// Tests for MONETRoof.FB_Roof's state machine (code review finding L5).
//
// Covers: the E_RoofState.unknown default before the first call, opening/closing (driven purely by
// Open()/Close()/SoftStop() and the ramp, no hardware inputs needed), stopped, and Reset() recovering
// from a cleared error.
//
// Deliberately not covered: the opened/closed states. Both need roof_limit_open/roof_limit_closed,
// which come from motors[i].opened/.closed -- AT%I*, hardware-linked, and this project configures no
// I/O. Validate those on the PLC instead (same as the plan's open step 5).
//
// Two things every test here has to do (without them FB_Roof never leaves the error / stopped state):
//  - SetDrivesOk(): FB_RoofMotor.motor_error is AT%I* and means "drive OK" (error := NOT motor_error). This project
//    maps no I/O, so it stays FALSE and both motors report error, which puts FB_Roof into the error state.
//  - one Call() before Open()/Close(): FB_Roof's parameters (max_speed, ...) are VAR_INPUTs that are only assigned
//    by a call, so Open() before the first call sets target_speed := TO_INT(0).
FUNCTION_BLOCK FB_Roof_State_Tests EXTENDS TcUnit.FB_TestSuite
VAR
END_VAR

Initial_State_Is_Unknown();
Open_Drives_State_To_Opening();
SoftStop_From_Moving_Drives_State_To_Stopped();
Close_Drives_State_To_Closing();
Reset_Clears_Error_State();

METHOD PRIVATE Call
VAR_IN_OUT
	roof		: MONETRoof.FB_Roof;
END_VAR
VAR_INPUT
	comm		: BROTLib.I_Comm;
END_VAR
roof(
	roof_number			:= 1,
	min_speed			:= 10000,
	max_speed			:= 30000,
	acceleration		:= 150,
	min_position		:= 0,
	max_position		:= 200,
	max_position_diff	:= 2,
	comm				:= comm);
END_METHOD

METHOD PRIVATE SetDrivesOk
VAR_IN_OUT
	roof		: MONETRoof.FB_Roof;
END_VAR
// motor_error is AT%I* with no I/O mapped here: TRUE = drive OK (see the header comment)
roof.motors[1].motor_error := TRUE;
roof.motors[2].motor_error := TRUE;
END_METHOD

METHOD PRIVATE Initial_State_Is_Unknown
VAR
	fbRoof	: MONETRoof.FB_Roof;
END_VAR
// Before FB_Roof is ever called, its VAR_OUTPUT members already hold their declared defaults.
TEST('Initial_State_Is_Unknown');
AssertTrue(Condition := fbRoof.state = E_RoofState.unknown, Message := 'declared default before the first call (was closed / enum value 0, L5)');
TEST_FINISHED();
END_METHOD

METHOD PRIVATE Open_Drives_State_To_Opening
VAR
	fbRoof	: MONETRoof.FB_Roof;
	fbComm	: FB_NullComm;
END_VAR
TEST('Open_Drives_State_To_Opening');
SetDrivesOk(roof := fbRoof);
Call(roof := fbRoof, comm := fbComm);	// assigns the parameters; Open() before this would see max_speed = 0
fbRoof.Open();
Call(roof := fbRoof, comm := fbComm);
AssertTrue(Condition := fbRoof.state = E_RoofState.opening, Message := 'speed > 0, both motors moving and direction_open: state becomes opening');
TEST_FINISHED();
END_METHOD

METHOD PRIVATE SoftStop_From_Moving_Drives_State_To_Stopped
VAR
	fbRoof	: MONETRoof.FB_Roof;
	fbComm	: FB_NullComm;
END_VAR
TEST('SoftStop_From_Moving_Drives_State_To_Stopped');
SetDrivesOk(roof := fbRoof);
Call(roof := fbRoof, comm := fbComm);	// assigns the parameters
fbRoof.Open();
Call(roof := fbRoof, comm := fbComm);
AssertTrue(Condition := fbRoof.state = E_RoofState.opening, Message := 'sanity: moving before the stop');
fbRoof.SoftStop();
// speed was 150, accel is 150: one ramp step reaches exactly 0
Call(roof := fbRoof, comm := fbComm);
AssertTrue(Condition := fbRoof.state = E_RoofState.stopped, Message := 'ramped down to 0, no longer moving, no switches engaged: stopped');
TEST_FINISHED();
END_METHOD

METHOD PRIVATE Close_Drives_State_To_Closing
VAR
	fbRoof	: MONETRoof.FB_Roof;
	fbComm	: FB_NullComm;
END_VAR
TEST('Close_Drives_State_To_Closing');
SetDrivesOk(roof := fbRoof);
Call(roof := fbRoof, comm := fbComm);	// assigns the parameters
fbRoof.Close();
Call(roof := fbRoof, comm := fbComm);
AssertTrue(Condition := fbRoof.state = E_RoofState.closing, Message := 'speed < 0, both motors moving and direction_close: state becomes closing');
TEST_FINISHED();
END_METHOD

METHOD PRIVATE Reset_Clears_Error_State
VAR
	fbRoof	: MONETRoof.FB_Roof;
	fbComm	: FB_NullComm;
END_VAR
TEST('Reset_Clears_Error_State');
SetDrivesOk(roof := fbRoof);
// invalid parameters (max_position = min_position) force config_error and the error state
fbRoof(roof_number := 1, min_speed := 10000, max_speed := 30000, acceleration := 150,
	min_position := 100, max_position := 100, max_position_diff := 2, comm := fbComm);
AssertTrue(Condition := fbRoof.state = E_RoofState.error, Message := 'sanity: config_error puts it in the error state');
fbRoof.Reset();
// same call as Call(), but spelled out: valid parameters now, and reset_roof is pending
Call(roof := fbRoof, comm := fbComm);
AssertFalse(Condition := fbRoof.config_error, Message := 'valid parameters now');
AssertTrue(Condition := fbRoof.state = E_RoofState.stopped, Message := 'reset_roof clears the latched error once the fault itself is gone');
TEST_FINISHED();
END_METHOD

END_FUNCTION_BLOCK

(* stored: Version 1.1.0.1, ProductVersion 3.1.4024.15
   POU FB_Roof_State_Tests: Id {cc5d60a7-7f07-4c34-b04e-da46caa01717}, SpecialFunc None
   Method Call: Id {c239d15f-3145-4b9a-8aa7-9aae42d1948c}
   Method SetDrivesOk: Id {3dba44f8-6f40-5d3a-8f2d-c2ce84c8a10b}
   Method Initial_State_Is_Unknown: Id {690883c6-9340-4841-8609-cea5e2d6306d}
   Method Open_Drives_State_To_Opening: Id {8cd11ade-06b1-445e-91e7-d122e282467e}
   Method SoftStop_From_Moving_Drives_State_To_Stopped: Id {7417f10f-cac2-4588-8139-3122a8cdd706}
   Method Close_Drives_State_To_Closing: Id {4ead5a6b-80a5-4455-bd68-94611f7a8ea8}
   Method Reset_Clears_Error_State: Id {1ca99bf6-322a-41b6-abda-0bd656922417} *)
